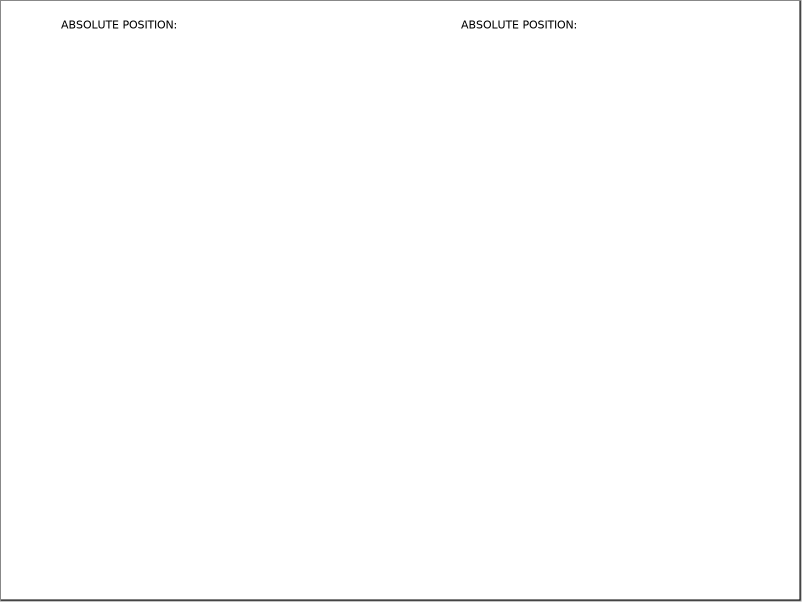
VISUALIZATION F13_Read_Actual_Velocity  // 802x602
    Rectangle (0,0 800x600)
    Label (10,10 170x30), "ABSOLUTE POSITION:"
    Label (410,10 170x30), "ABSOLUTE POSITION:"
END_VISUALIZATION

(* stored: Version 1.1.0.1, ProductVersion 3.1.4022.7
   Visu F13_Read_Actual_Velocity: Id {f2b4dbf4-308c-4edc-8c0a-afb9b04d0f2c} *)
